FUNCTION_BLOCK FB_SAstiffness
VAR_INPUT
	cycles : INT := 0;
END_VAR
VAR_OUTPUT
	cyclesOut : INT := 0;
	force : REAL := 0;
END_VAR
VAR
	counter : INT := 0;
	sign : REAL := 1;
END_VAR

counter := counter + 1;

IF counter = 50 THEN
	force := force + sign;
	counter := 0;
END_IF

IF force = 500 THEN
	sign := -1;
	cycles := cycles + 1;
END_IF

IF force = -500 THEN
	sign := 1;
	cycles := cycles + 1;
END_IF

cyclesOut := cycles;

END_FUNCTION_BLOCK

(* stored: Version 1.1.0.1, ProductVersion 3.1.4024.12
   POU FB_SAstiffness: Id {0554bc39-3a5f-4c1e-b75b-b43e140973bf}, SpecialFunc None *)
